{attribute addProperty BoxType "EJ3004-0000-0020"}
{attribute addProperty Id "AI_Standard_ChannelAT %I*ARRAY[0..3] OF AI_Standard_Channel_E1AC0F6232440.50WcStateAT %I*WcState_98A4DF7520.250InfoDataAT %I*InfoData_BC63D37F80100"}
{attribute addProperty CRC "2350437303"}
{attribute addProperty SizeInBites "406"}
{attribute addProperty SizeInBytes "50.75"}
TYPE EJ3004_19668D28 :
STRUCT
	{attribute addProperty Name "AI_Standard_Channel"}
	AI_Standard_Channel : ARRAY[0..3] OF AI_Standard_Channel_E1AC0F62;
	{attribute addProperty Name "WcState"}
	WcState : WcState_98A4DF75;
	{attribute addProperty Name "InfoData"}
	InfoData : InfoData_BC63D37F;
END_STRUCT
END_TYPE

(* stored: Version 1.2.0.0, ProductVersion 3.1.4024.9
   DUT EJ3004_19668D28: Id {220f03b7-5cfe-47bd-ab9d-b0725099e98d} *)
